TYPE ST_PostRunReport :
STRUCT
	runNo				: INT;
	methodName			: STRING(100);
	methodRevision		: STRING(100);
	methodCreatedBy		: STRING(100);
	methodCreatedOn		: STRING(100);
	solvent_R1			: STRING(100);
	solvent_R2			: STRING(100);
	solvent_W1			: STRING(100);
	solvent_W2			: STRING(100);
	time_R1				: STRING(100);
	time_R2				: STRING(100);
	time_W1				: STRING(100);
	time_W2				: STRING(100);
	velocity_R1			: STRING(100);
	velocity_R2			: STRING(100);
	velocity_W1			: STRING(100);
	velocity_W2			: STRING(100);
	soakTime			: STRING(100);
	agitate_1_Time		: STRING(100);
	agitate_2_Time		: STRING(100);
	vialsToFill			: STRING(100);
	vialPrimeVol		: STRING(100);
	vial_1_FillVol		: STRING(100);
	vial_2_4_FillVol	: STRING(100);
	airDryTime			: STRING(100);
	analyst				: STRING(100);
	calibrationNo		: STRING(100);
	comment				: STRING(100);
	softwareVersion		: STRING(100);
	sysMasterRevision	: STRING(100);
	sysSettingsRevision	: STRING(100);
	meterVelocity		: STRING(100);
	runVelocity			: STRING(100);
	emptyTubesFactor	: STRING(100);
	fillTubesFactor		: STRING(100);
	solvent1NameRevision: STRING(100);
	solvent2NameRevision: STRING(100);
	solvent3NameRevision: STRING(100);
	solvent4NameRevision: STRING(100);
	timeEventStarted	: STRING(100);
	timeEventCompleted	: STRING(100);
END_STRUCT
END_TYPE

(* stored: Version 1.1.0.1, ProductVersion 3.1.4024.12
   DUT ST_PostRunReport: Id {f2068320-89cd-429f-819a-3a8eabf602d9} *)
